TYPE Datastructure1 :
STRUCT
	Name : STRING(255);
	Result : BOOL;
END_STRUCT
END_TYPE

(* stored: Version 1.1.0.1, ProductVersion 3.1.4024.10
   DUT Datastructure1: Id {218c29dd-b2a6-4335-93b6-ae77c2a9207a} *)
